// TwinCAT 3 PLC project MAS418
// ProgramVersion: 3.1.4023.0
// libraries:
//   Tc2_Standard, * (Beckhoff Automation GmbH)
//   Tc2_System, * (Beckhoff Automation GmbH)
//   Tc3_Module, * (Beckhoff Automation GmbH)
// project tree:
//   Actuators/FBs/ FB_AutoCyl.TcPOU, FB_autoWinch.TcPOU, FB_ClosedLoopControl.TcPOU, FB_Manual.TcPOU, FB_MotionReferenceGenerator.TcPOU, FB_OpenLoopControlCyl.TcPOU, FB_ResetIntegralController.TcPOU, FB_Timer.TcPOU, FB_OpenLoopWinchControl.TcPOU
//   Actuators/GVLs/ G_ControlParameters.TcGVL, G_Parameters.TcGVL
//   Actuators/Programs/ P_ControlSystem.TcPOU
//   Actuators/Structs/ ST_AutoControllerSelection.TcDUT, ST_ClosedLoopParams.TcDUT, ST_CylinderParameters.TcDUT, ST_MotionReferenceParams.TcDUT, ST_OpenLoopParams.TcDUT, ST_ScalingParameters.TcDUT, ST_SetControlParams.TcDUT, ST_ValveDeadband.TcDUT, ST_WinchParameters.TcDUT
//   / GlobalTextList.TcGTLO, PlcTask.TcTTO, Visualization Manager.TcVMO (not stored)
//   HMI/ CtrlBox.TcVIS, P_VHMI.TcPOU, VirtualBoxHMI.TcVIS
//   HMI/Enums/ E_Mode.TcDUT, E_Status.TcDUT, I_Mode.TcIO
//   HMI/FBs/ FB_Mode.TcPOU, FB_Status.TcPOU
//   HMI/GVLs/ G_Modes.TcGVL
//   HMI/Structs/ ST_VisuParam.TcDUT
//   Inputs/FBs/ FB_Encoder.TcPOU, FB_FlowScaling.TcPOU, FB_JoystickScale.TcPOU, FB_Scaling.TcPOU
//   Inputs/GVLs/ G_InputsRaw.TcGVL, G_InputsScaled.TcGVL, G_StructData.TcGVL
//   Inputs/Programs/ P_ScaleSensors.TcPOU
//   Inputs/Structs/ ST_FlowScale.TcDUT, ST_InputScaling.TcDUT, ST_JoystickScale.TcDUT
//   Outputs/FBs/ FB_ValveOutput.TcPOU
//   Outputs/GVLs/ G_Outputs.TcGVL
//   Outputs/Programs/ P_out.TcPOU
//   Outputs/Structs/ ST_ValveOutput.TcDUT
//   POUs/ MAIN.TcPOU
// real-time tasks:
//   TASK PlcTask: cycle T#10ms, priority 20, ADS port 350
// I/O:
//   DEVICE Device 1 (EtherCAT) (disabled), AmsNetId 169.254.36.244.2.1
//     Term 1 (EK1100) [EK1100 EtherCAT Coupler (2A E-Bus)]
//       Term 2 (EL1008)
//       Term 3 (EL2008)
//       Term 4 (EL3068)
//       Term 5 (EL3068) [EL3068 8Ch. Ana. Input 0-10V]
//       Term 6 (EL3174) [EL3174 4Ch. Ana. Input +/-10V Diff., +/-20mA SingleEnded, 16 Bit]
//       Term 7 (EL3255)
//       Term 8 (EL4104)
//       Term 9 (EL9011)
//     Box 10 (Fraba EtherCAT) [Absolute Rotary Encoder IXARC V01.05]
// variable links:
//   MAS418 Instance <-> Device 1 (EtherCAT)/Box 10 (Fraba EtherCAT)
//     PlcTask Inputs/G_InputsRaw.nEncoderValue <-> Encoder/Position Value
//   MAS418 Instance <-> Device 1 (EtherCAT)/Term 1 (EK1100)/Term 2 (EL1008)
//     PlcTask Inputs/G_InputsRaw.bJoyTopSwitch <-> Channel 5/Input
//     PlcTask Inputs/G_InputsRaw.bSelectAuto <-> Channel 2/Input
//     PlcTask Inputs/G_InputsRaw.bSelectManual <-> Channel 1/Input
//     PlcTask Inputs/G_InputsRaw.bStartButton <-> Channel 3/Input
//     PlcTask Inputs/G_InputsRaw.bStopButton <-> Channel 4/Input
//   MAS418 Instance <-> Device 1 (EtherCAT)/Term 1 (EK1100)/Term 3 (EL2008)
//     PlcTask Outputs/G_Outputs.bGreenLight <-> Channel 1/Output
//     PlcTask Outputs/G_Outputs.bRedLight <-> Channel 2/Output
//     PlcTask Outputs/G_Outputs.stCylinderOutputs.bEnable <-> Channel 4/Output
//     PlcTask Outputs/G_Outputs.stWinchOutputs.bEnable <-> Channel 3/Output
//   MAS418 Instance <-> Device 1 (EtherCAT)/Term 1 (EK1100)/Term 4 (EL3068)
//     PlcTask Inputs/G_InputsRaw.nPistonPressure <-> AI Standard Channel 4/Value
//     PlcTask Inputs/G_InputsRaw.nReturnPressure <-> AI Standard Channel 2/Value
//     PlcTask Inputs/G_InputsRaw.nRodPressure <-> AI Standard Channel 3/Value
//     PlcTask Inputs/G_InputsRaw.nSupplyPressure <-> AI Standard Channel 1/Value
//     PlcTask Inputs/G_InputsRaw.nWinch_A1_Pressure <-> AI Standard Channel 5/Value
//     PlcTask Inputs/G_InputsRaw.nWinch_A_Pressure <-> AI Standard Channel 7/Value
//     PlcTask Inputs/G_InputsRaw.nWinch_B1_Pressure <-> AI Standard Channel 6/Value
//     PlcTask Inputs/G_InputsRaw.nWinch_B_Pressure <-> AI Standard Channel 8/Value
//   MAS418 Instance <-> Device 1 (EtherCAT)/Term 1 (EK1100)/Term 5 (EL3068)
//     PlcTask Inputs/G_InputsRaw.nWinchDrainPressure <-> AI Standard Channel 1/Value
//   MAS418 Instance <-> Device 1 (EtherCAT)/Term 1 (EK1100)/Term 6 (EL3174)
//     PlcTask Inputs/G_InputsRaw.nWinchFlow <-> AI Standard Channel 1/Value
//   MAS418 Instance <-> Device 1 (EtherCAT)/Term 1 (EK1100)/Term 7 (EL3255)
//     PlcTask Inputs/G_InputsRaw.nJoyCyl <-> AI Standard Channel 2/Value
//     PlcTask Inputs/G_InputsRaw.nJoyWinch <-> AI Standard Channel 3/Value
//     PlcTask Inputs/G_InputsRaw.nPositionCylPiston <-> AI Standard Channel 1/Value
//   MAS418 Instance <-> Device 1 (EtherCAT)/Term 1 (EK1100)/Term 8 (EL4104)
//     PlcTask Outputs/G_Outputs.stCylinderOutputs.nValveOutput <-> AO Output Channel 2/Analog output
//     PlcTask Outputs/G_Outputs.stWinchOutputs.nValveOutput <-> AO Output Channel 1/Analog output

CONFIGURATION MAS418
    RESOURCE PLC ON TwinCAT3
        TASK PlcTask(INTERVAL := T#10ms, PRIORITY := 20);
        PROGRAM MAIN WITH PlcTask : MAIN;
    END_RESOURCE
END_CONFIGURATION

// ---- Actuators/Structs/ST_AutoControllerSelection.TcDUT
TYPE ST_AutoControllerSelection :
STRUCT
	bStartFeedForward : BOOL;
	bStartClosedLoop : BOOL;
	bEnableIntegral : BOOL; 
	
END_STRUCT
END_TYPE

// ---- Actuators/Structs/ST_ClosedLoopParams.TcDUT
TYPE ST_ClosedLoopParams :
STRUCT
	fProportionalGain: LREAL;
	fIntegralGain: LREAL;
	fMaxAllowableError : LREAL; 
END_STRUCT
END_TYPE

// ---- Actuators/Structs/ST_CylinderParameters.TcDUT
TYPE ST_CylinderParameters :
STRUCT
	fCylMaxSpeed : LREAL := 0.05; // m/s
END_STRUCT
END_TYPE

// ---- Actuators/Structs/ST_MotionReferenceParams.TcDUT
TYPE ST_MotionReferenceParams :
STRUCT
	fStartPosition_m: LREAL := 0.0;
	fStartVelocity_m: LREAL := 0.0;
	fPositionSetpoint_m: LREAL := 0.2;
	fVelocitySetpoint_m: LREAL := 0.02;
	fTimeBeforeStarting_s: LREAL := 1.5;
	fRampTime_s: LREAL := 2.0;
	fHoldPositionTime_s: LREAL := 4.0;
	
	// Saturation
	fMaxPosition 			: LREAL := 0.6;
	fMinPosition 			: LREAL := 0.0;
	fMaxVelocity 			: LREAL := 0.04;
	
	// Cycle time
	fCycleTime : LREAL := 0.001; // Same as matlab/simulink
END_STRUCT
END_TYPE

// ---- Actuators/Structs/ST_OpenLoopParams.TcDUT
TYPE ST_OpenLoopParams :
STRUCT
	fBoresideArea : LREAL;
	fAnnulusArea : LREAL; 
	fMaxFlow : LREAL; 
END_STRUCT
END_TYPE

// ---- Actuators/Structs/ST_ScalingParameters.TcDUT
TYPE ST_ScalingParameters :
STRUCT
	stCylPos : ST_InputScaling := (fMaxInputValue := 32295.0, fMinInputValue := 229.0, fMaxOutputValue := 0.5, fMinOutputValue := 0.0);
	stPressure400bar 	: ST_InputScaling := (fMaxInputValue := 32767.0, fMinInputValue := 0.0, fMaxOutputValue := 400.0, fMinOutputValue := 0.0);
	stPressure40bar 	: ST_InputScaling := (fMaxInputValue := 32767.0, fMinInputValue := 0.0, fMaxOutputValue := 40.0, fMinOutputValue := 0.0);
	stFlow : ST_FlowScale := (fMaxFlowInput := 32295.0, fMinFlowInput := 0.0, fNeutralFlowInput := 15450, fNeutralDeadband := 50.0, fMaxFlowOutput := 150.0, fMinFlowOutput := -150.0, fNeutralFlowOutput := 0.0);
END_STRUCT
END_TYPE

// ---- Actuators/Structs/ST_SetControlParams.TcDUT
TYPE ST_SetControlParams :
STRUCT
	stWinchControlClosedSettings : ST_ClosedLoopParams :=(fProportionalGain:=10, fIntegralGain:=5, fMaxAllowableError := 0.01);
	stCylControlCloesSettings : ST_ClosedLoopParams :=(fProportionalGain:=10, fIntegralGain:=5, fMaxAllowableError := 0.01);
	stWinchControlOpenSettings : ST_OpenLoopParams :=(fBoresideArea:=0.0033183, fAnnulusArea:=0.0023562, fMaxFlow:=150*0.5);
	stCylControlOpenSettings : ST_OpenLoopParams :=(fBoresideArea:=0, fAnnulusArea:=0, fMaxFlow:=150*0.5); 
END_STRUCT
END_TYPE

// ---- Actuators/Structs/ST_ValveDeadband.TcDUT
TYPE ST_ValveDeadband :
STRUCT
	fPosMax	: LREAL := 29490.0; 
	fPosMin	: LREAL := 20950.0; 
	fNegMin : LREAL := 18250.0; 
	fNegMax	: LREAL := 9830.0; 
END_STRUCT
END_TYPE

// ---- Actuators/Structs/ST_WinchParameters.TcDUT
TYPE ST_WinchParameters :
STRUCT
	fEncoderOffset : LREAL := 17574.8;
	fWinchDrumScaling : LREAL := 0.000744309;
	fWinchMotorDisplacement : LREAL := 32.0; 
	fWinchMaxSpeed : LREAL := 0.05; // rad/s
	
END_STRUCT
END_TYPE

// ---- HMI/Enums/E_Mode.TcDUT
{attribute 'qualified_only'}
{attribute 'strict'}
TYPE E_Mode :
(
	OFF := 0,
	Auto := 1,
	Manual :=2
);
END_TYPE

// ---- HMI/Enums/E_Status.TcDUT
{attribute 'qualified_only'}
{attribute 'strict'}
TYPE E_Status :
(	NotReady := 0,
	Ready := 1,
	Starting := 2,
	Running := 3,
	Stopping := 4,
	Fault := 5,
	JoyStick := 6
);
END_TYPE

// ---- HMI/Structs/ST_VisuParam.TcDUT
TYPE ST_VisuParam :
STRUCT
bOn : BOOL;
bAuto : BOOL;
bStart : BOOL;
bStop : BOOL;
bRunning : BOOL;
bFault : BOOL;
fJoy_X : REAL;
fJoy_Y : REAL;
bTopSwitchJoy : BOOL;
END_STRUCT
END_TYPE

// ---- Inputs/Structs/ST_FlowScale.TcDUT
TYPE ST_FlowScale :
STRUCT
	fMaxFlowInput : LREAL; 
	fMinFlowInput : LREAL;
    fNeutralFlowInput : LREAL; 
	fNeutralDeadband : LREAL; 
	fMaxFlowOutput : LREAL; 
	fMinFlowOutput : LREAL; 
	fNeutralFlowOutput : LREAL; 
END_STRUCT
END_TYPE

// ---- Inputs/Structs/ST_InputScaling.TcDUT
TYPE ST_InputScaling :
STRUCT
	fMaxInputValue : LREAL;
	fMinInputValue : LREAL;
	fMaxOutputValue : LREAL;
	fMinOutputValue : LREAL; 
END_STRUCT
END_TYPE

// ---- Inputs/Structs/ST_JoystickScale.TcDUT
TYPE ST_JoystickScale :
STRUCT
	fMaxInputValue : LREAL := 20509.0;
	fMinInputValue : LREAL  := 11787.0; 
	fNeutralInputValue : LREAL  := 16175; 
	fNeutralDeadband : LREAL  := 50.0; 
	fMaxOutputValue : LREAL  := 1.0; 
	fMinOutputValue : LREAL  := -1.0;
	fNeutralOutputValue : LREAL  := 0.0; 
END_STRUCT
END_TYPE

// ---- Outputs/Structs/ST_ValveOutput.TcDUT
TYPE ST_ValveOutput :
STRUCT
	bEnable					AT %Q* : BOOL := 0;
	nValveOutput 			AT %Q* : INT := 19660; // Initial value at offset
END_STRUCT
END_TYPE

// ---- Actuators/GVLs/G_ControlParameters.TcGVL
{attribute 'qualified_only'}
VAR_GLOBAL
	bWinchEnable : BOOL;
	bCylEnable : BOOL;
	
	// Parameters for control circuit
	fWinch_ControlInput : LREAL;
	fWinchTimer	: LREAL;
	fCylinder_ControlInput : LREAL;
	fCylTimer : LREAL;
	fControlSignal_Winch : LREAL;
	fControlSignal_Cyl : LREAL; 
	
	// Reference signals / Setpoints
	fVelRefWinch : LREAL;
	fPosRefWinch : LREAL;
	fVelRefCyl : LREAL;
	fPosRefCyl : LREAL;
	fPosErrorWinch : LREAL;
	fPosErrorCyl : LREAL; 
	
	bDeadBandCompOn : BOOL := TRUE; 
END_VAR

// ---- Actuators/GVLs/G_Parameters.TcGVL
{attribute 'qualified_only'}
VAR_GLOBAL
	stCylParams : ST_CylinderParameters;
	stValve : ST_ValveDeadband;
	stWinchParams : ST_WinchParameters; 
	stCommonScaling : ST_ScalingParameters; 
	stControl : ST_SetControlParams;  
END_VAR

// ---- HMI/GVLs/G_Modes.TcGVL
{attribute 'qualified_only'}
VAR_GLOBAL
	bManualMode : BOOL;
	bAutoMode : BOOL; 
	bStart : BOOL;
	bStop : BOOL;
	bSwitch : BOOL; 
	bCylEnable : BOOL;
	bWinchEnable : BOOL; 
	bOn : BOOL; 
	stMotionRefWinch : ST_MotionReferenceParams;
	stMotionRefCyl : ST_MotionReferenceParams;
	stCylinderControl : ST_AutoControllerSelection;
	stWinchControl : ST_AutoControllerSelection; 
	eStatus : E_Status;
	eMode : E_Mode; 
	stVisualParams : ST_VisuParam; 
END_VAR

// ---- Inputs/GVLs/G_InputsRaw.TcGVL
{attribute 'qualified_only'}
VAR_GLOBAL
	bSelectOff AT %I* : BOOL; 
	bSelectManual	AT %I* : BOOL;
	bSelectAuto AT %I* : BOOL;
	bStartButton AT %I* : BOOL;
	bStopButton	AT %I* : BOOL;
	bJoyTopSwitch	AT %I* : BOOL;
	
	// Joystick
	nJoyCyl AT %I* : INT; 					
	nJoyWinch AT %I* : INT; 	

	// Encoder					
	nPositionCylPiston AT %I* : INT; 		
	nEncoderValue AT %I* : UDINT;
		
	
	// Pressures Valve x Cyl
	nSupplyPressure AT %I* : INT;
	nReturnPressure AT %I* : INT;
	nPistonPressure AT %I* : INT;
	nRodPressure AT %I* : INT; 
	
	// Pressures Winch
	nWinch_A_Pressure AT %I* : INT;
	nWinch_A1_Pressure AT %I* : INT;
	nWinch_B_Pressure AT %I* : INT;
	nWinch_B1_Pressure AT %I* : INT;
	nWinchDrainPressure AT %I* : INT; 

	// Winch flow
	nWinchFlow AT %I* : INT; 		
END_VAR

// ---- Inputs/GVLs/G_InputsScaled.TcGVL
{attribute 'qualified_only'}
VAR_GLOBAL
	
	// Joystick
	fJoystickScaledX 		: LREAL;
	fJoystickScaledY 		: LREAL;
	
	// Cylinder and winch position
	fCylPosition : LREAL;	
	fEncoderPosition : LREAL;
	fWirePosition : LREAL;
	
	// Pressures Valve
	fSupplyPressure			: LREAL;
	fReturnPressure 			: LREAL;
	
	// Pressures Cylinder
	fPistonPressure 	: LREAL;
	fRodPressure		: LREAL;
	
	// Pressures Winch
	fWinch_A_Pressure 		: LREAL;
	fWinch_A1_Pressure 		: LREAL;
	fWinch_B_Pressure	: LREAL;
	fWinch_B1_Pressure	: LREAL;
	fWinchDrainPressure			: LREAL;
	
	// Winch Flow
	fWinchFlow 					: LREAL;
END_VAR

// ---- Inputs/GVLs/G_StructData.TcGVL
{attribute 'qualified_only'}
VAR_GLOBAL
	stJoystickX : ST_JoystickScale;
	stJoystickY : ST_JoystickScale; 
	stInputs : ST_InputScaling;
	stFlows : ST_FlowScale;
END_VAR

// ---- Outputs/GVLs/G_Outputs.TcGVL
{attribute 'qualified_only'}
VAR_GLOBAL
	bGreenLight AT %Q* : BOOL;
	bRedLight AT %Q* : BOOL;
	
	stWinchOutputs : ST_ValveOutput;
	stCylinderOutputs : ST_ValveOutput; 
END_VAR

// ---- HMI/Enums/I_Mode.TcIO

INTERFACE I_Mode

METHOD Auto
VAR_INPUT
	bEnable : BOOL;
END_VAR
END_METHOD

METHOD Manual
VAR_INPUT
	bEnable : BOOL;
END_VAR
END_METHOD

METHOD OFF 
VAR_INPUT
	bEnable : BOOL;
END_VAR
END_METHOD

END_INTERFACE

// ---- POUs/MAIN.TcPOU
PROGRAM MAIN
VAR
END_VAR

P_ScaleSensors();
P_out();
P_VHMI();
P_ControlSystem();

END_PROGRAM

// ---- Inputs/Programs/P_ScaleSensors.TcPOU
PROGRAM P_ScaleSensors
VAR
	// Joystick
	fbJoystickX : FB_JoystickScale;
	fbJoystickY : FB_JoystickScale;
	
	// Positions
	fbWinchPosition : FB_Encoder;
	fbCylPosition : FB_Scaling;
	
	// Pressures
	fbSupplyPressure : FB_Scaling;
	fbReturnPressure : FB_Scaling;
	fbPistonPressure : FB_Scaling;
	fbRodPressure	: FB_Scaling;
	fbWinch_A_Pressure : FB_Scaling;
	fbWinch_A1_Pressure : FB_Scaling;
	fbWinch_B_Pressure : FB_Scaling;
	fbWinch_B1_Pressure : FB_Scaling;
	fbWinchDrainPressure : FB_Scaling;
	
	// Flows
	fbWinchFlow	: FB_FlowScaling;
END_VAR

// Scaling Joystick
fbJoystickX(bEnable := G_Modes.bManualMode, nRawInput := G_InputsRaw.nJoyCyl,
	fNormalizedOutput => G_InputsScaled.fJoystickScaledX);

fbJoystickY(bEnable := G_Modes.bManualMode, 
	nRawInput := G_InputsRaw.nJoyWinch, 
	fNormalizedOutput => G_InputsScaled.fJoystickScaledY);
 
// Winch position & Cylinder position
fbWinchPosition (
	nRawInput := G_InputsRaw.nEncoderValue, 
	fPosition => G_InputsScaled.fEncoderPosition,
	fWirePosition => G_InputsScaled.fWirePosition);

fbCylPosition(
	nRawInput := G_InputsRaw.nPositionCylPiston,
	stInputScaling := G_Parameters.stCommonScaling.stCylPos,
	fScaledOutput => G_InputsScaled.fCylPosition);


// Pressures

fbSupplyPressure(
	nRawInput := G_InputsRaw.nSupplyPressure,
	stInputScaling := G_Parameters.stCommonScaling.stPressure400bar,
	fScaledOutput => G_InputsScaled.fSupplyPressure);

fbReturnPressure(
	nRawInput := G_InputsRaw.nReturnPressure,
	stInputScaling := G_Parameters.stCommonScaling.stPressure40bar,
	fScaledOutput => G_InputsScaled.fReturnPressure);

fbPistonPressure(
	nRawInput := G_InputsRaw.nPistonPressure,
	stInputScaling := G_Parameters.stCommonScaling.stPressure400bar,
	fScaledOutput => G_InputsScaled.fPistonPressure);
	
fbRodPressure(
	nRawInput := G_InputsRaw.nRodPressure,
	stInputScaling := G_Parameters.stCommonScaling.stPressure400bar,
	fScaledOutput => G_InputsScaled.fRodPressure);
	
fbWinch_A_Pressure(
	nRawInput := G_InputsRaw.nWinch_A_Pressure,
	stInputScaling := G_Parameters.stCommonScaling.stPressure400bar,
	fScaledOutput => G_InputsScaled.fWinch_A_Pressure); 
	
fbWinch_A1_Pressure(
	nRawInput := G_InputsRaw.nWinch_A1_Pressure,
	stInputScaling := G_Parameters.stCommonScaling.stPressure400bar,
	fScaledOutput => G_InputsScaled.fWinch_A1_Pressure);

fbWinch_B_Pressure(
	nRawInput := G_InputsRaw.nWinch_B_Pressure,
	stInputScaling := G_Parameters.stCommonScaling.stPressure400bar,
	fScaledOutput => G_InputsScaled.fWinch_B_Pressure);

fbWinch_B1_Pressure(
	nRawInput := G_InputsRaw.nWinch_B1_Pressure,
	stInputScaling := G_Parameters.stCommonScaling.stPressure400bar,
	fScaledOutput => G_InputsScaled.fWinch_B1_Pressure);
	
fbWinchDrainPressure(
	nRawInput := G_InputsRaw.nWinchDrainPressure,
	stInputScaling := G_Parameters.stCommonScaling.stPressure40bar,
	fScaledOutput => G_InputsScaled.fWinchDrainPressure);

fbWinchFlow(
	nRawInput := G_InputsRaw.nWinchFlow,
	stFlowParams := G_Parameters.stCommonScaling.stFlow,
	fScaledFlow => G_InputsScaled.fWinchFlow);

END_PROGRAM

// ---- Inputs/FBs/FB_JoystickScale.TcPOU
FUNCTION_BLOCK FB_JoystickScale
VAR_INPUT
	bEnable 				: BOOL;
	nRawInput 				: INT;
END_VAR
VAR_OUTPUT
	fNormalizedOutput 		: LREAL;
END_VAR
VAR
	stJoystickScale  : ST_JoystickScale;
	fRawInput 				: LREAL;
	fTempInput 				: LREAL;
	fTempOutput 			: LREAL;
END_VAR

fRawInput := INT_TO_LREAL(nRawInput);

fTempInput := fRawInput - stJoystickScale.fNeutralInputValue;

IF fTempInput > stJoystickScale.fNeutralDeadband THEN
	fTempOutput := fTempInput/(stJoystickScale.fMaxInputValue - stJoystickScale.fNeutralInputValue);
ELSIF fTempInput < -stJoystickScale.fNeutralDeadband THEN	
	fTempOutput := fTempInput/(stJoystickScale.fNeutralInputValue - stJoystickScale.fMinInputValue);
ELSE
	fTempOutput := 0.0;
END_IF

IF NOT(bEnable) THEN
	fNormalizedOutput := 0.0;
ELSE
	fNormalizedOutput := LIMIT(stJoystickScale.fMinOutputValue, fTempOutput, stJoystickScale.fMaxOutputValue);
END_IF

END_FUNCTION_BLOCK

// ---- Inputs/FBs/FB_Encoder.TcPOU
FUNCTION_BLOCK FB_Encoder
VAR_INPUT
	nRawInput : UDINT;
	stParam 		: ST_WinchParameters; 
END_VAR
VAR_OUTPUT
	fPosition 		: LREAL;
	fWirePosition : LREAL; 
END_VAR
VAR PERSISTENT
	nRounds			: DINT;
	nRawLast 		: DINT;
END_VAR	
VAR
	nInput 		: DINT;
	nTempInputDiff	: DINT;
	nCount 			: DINT;
	nMaxValue30bit 	: DINT :=  1073741823; // 2^30 - 1	
	nThreshold30bit	: DINT := nMaxValue30bit/2;
	fScale16bit		: LREAL := 360.0/65535.0; // 360deg/(2^16 - 1)
	fTempPosition   : LREAL;
END_VAR

// Convert to DINT (same as const values)
nInput := UDINT_TO_DINT(nRawInput);

// Define Encoder Rounds
nTempInputDiff := nInput - nRawLast;
IF (nTempInputDiff > nThreshold30bit) THEN
	nRounds := nRounds - 1;
END_IF

IF (nTempInputDiff < -nThreshold30bit) THEN
	nRounds := nRounds + 1;
END_IF

// Count Encoder Rounds
nCount := nInput + nRounds*nMaxValue30bit;

//Position Output
fPosition := DINT_TO_LREAL(nCount)*fScale16bit - stParam.fEncoderOffset; // Encoder position
fWirePosition := fPosition * G_Parameters.stWinchParams.fWinchDrumScaling; // WIre position

END_FUNCTION_BLOCK

// ---- Inputs/FBs/FB_Scaling.TcPOU
FUNCTION_BLOCK FB_Scaling
VAR_INPUT
	nRawInput : INT; 
	stInputScaling : ST_InputScaling; 
END_VAR
VAR_OUTPUT
	fScaledOutput : LREAL;

END_VAR
VAR
	fRawInput : LREAL;
	fNormInput : LREAL;
	
END_VAR

fRawInput := INT_TO_LREAL(nRawInput);

fNormInput := (fRawInput - stInputScaling.fMinInputValue) / (stInputScaling.fMaxInputValue - stInputScaling.fMinInputValue);

fScaledOutput := LIMIT(stInputScaling.fMinOutputValue, stInputScaling.fMinOutputValue + fNormInput*(stInputScaling.fMaxOutputValue - stInputScaling.fMinOutputValue), stInputScaling.fMaxOutputValue);

END_FUNCTION_BLOCK

// ---- Inputs/FBs/FB_FlowScaling.TcPOU
FUNCTION_BLOCK FB_FlowScaling
VAR_INPUT
	nRawInput : INT;
	stFlowParams : ST_FlowScale; 
END_VAR
VAR_OUTPUT
	fScaledFlow : LREAL; 
END_VAR
VAR
	fRawInput 				: LREAL;
	fTempInput 				: LREAL;
	fTempOutput 			: LREAL;
END_VAR

fRawInput := INT_TO_LREAL(nRawInput);

fTempInput := fRawInput - stFlowParams.fNeutralFlowInput;

IF fTempInput > stFlowParams.fNeutralDeadband THEN
	fTempOutput := fTempInput/(stFlowParams.fMaxFlowInput - stFlowParams.fNeutralFlowInput);
ELSIF fTempInput < -stFlowParams.fNeutralDeadband THEN	
	fTempOutput := fTempInput/(stFlowParams.fNeutralFlowInput - stFlowParams.fMinFlowInput);
ELSE
	fTempOutput := 0.0;
END_IF

fScaledFlow := LIMIT(stFlowParams.fMinFlowOutput, fTempOutput*150.0, stFlowParams.fMaxFlowOutput);

END_FUNCTION_BLOCK

// ---- Outputs/Programs/P_out.TcPOU
PROGRAM P_out
VAR
	fbWinchOutput 		: FB_ValveOutput;
	fbCylOutput 		: FB_ValveOutput;
END_VAR

// Settings to ensure output if either auto or manual is selected:
G_Outputs.stWinchOutputs.bEnable := G_Modes.bAutoMode OR G_Modes.bManualMode; 
G_Outputs.stCylinderOutputs.bEnable := G_Modes.bAutoMode OR G_Modes.bManualMode; 


fbWinchOutput(bEnable := G_ControlParameters.bWinchEnable OR G_ControlParameters.fWinchTimer > 0.0,
	bDeadBandCompOn := G_ControlParameters.bDeadBandCompOn,
	stValveDeadBand := G_Parameters.stValve,
	fNormalizedInput := G_ControlParameters.fWinch_ControlInput,
	nOutput => G_Outputs.stWinchOutputs.nValveOutput); 
	
	
fbCylOutput(bEnable := G_ControlParameters.bWinchEnable OR G_ControlParameters.fCylTimer > 0.0,
	bDeadBandCompOn := G_ControlParameters.bDeadBandCompOn,
	stValveDeadBand := G_Parameters.stValve,
	fNormalizedInput := G_ControlParameters.fCylinder_ControlInput,
	nOutput => G_Outputs.stCylinderOutputs.nValveOutput);

END_PROGRAM

// ---- Outputs/FBs/FB_ValveOutput.TcPOU
FUNCTION_BLOCK FB_ValveOutput
VAR_INPUT
	bEnable 			: BOOL;
	bDeadBandCompOn 	: BOOL;
	stValveDeadBand 	: ST_ValveDeadBand;
	fNormalizedInput 	: LREAL;
END_VAR
VAR_OUTPUT
	bEnableValveOutput : BOOL;
	nOutput : INT; 
END_VAR
VAR
	nOffset 	: INT := 19660;
	nMaxValue	: INT := 29490;
	nMinValue 	: INT :=  9830;
	nTempOutput : INT;
END_VAR

IF	bDeadBandCompOn THEN
	IF fNormalizedInput > 0.0 THEN
		nTempOutput := LREAL_TO_INT(ABS(fNormalizedInput*(stValveDeadBand.fPosMax - stValveDeadBand.fPosMin) + stValveDeadBand.fPosMin));
	ELSIF fNormalizedInput < 0.0 THEN
		nTempOutput := LREAL_TO_INT(ABS(fNormalizedInput*(stValveDeadBand.fNegMax - stValveDeadBand.fNegMin) - stValveDeadBand.fNegMin));
	ELSE
		nTempOutput := nOffset;
	END_IF
ELSE
	IF fNormalizedInput > 0.0 THEN
		nTempOutput := LREAL_TO_INT(ABS(fNormalizedInput*(32767.0 - 19660.0) + 19660.0));
	ELSIF fNormalizedInput < 0.0 THEN
		nTempOutput := LREAL_TO_INT(ABS(fNormalizedInput*(0 - 19660.0) - 19660.0));
	ELSE
		nTempOutput := nOffset;
	END_IF	
END_IF	

IF bEnable THEN
	nOutput := LIMIT(nMinValue, nTempOutput, nMaxValue);
	bEnableValveOutput := TRUE; 
ELSE 	
	nOutput := nOffset;
	bEnableValveOutput := FALSE;	
END_IF

END_FUNCTION_BLOCK

// ---- HMI/P_VHMI.TcPOU
PROGRAM P_VHMI
VAR
	fbModeSelect : FB_Mode;
END_VAR

fbModeSelect(
	bMode := G_Modes.bAutoMode);

END_PROGRAM

// ---- HMI/FBs/FB_Mode.TcPOU
FUNCTION_BLOCK FB_Mode
VAR_INPUT
	bMode : BOOL; 
END_VAR
VAR_OUTPUT
	
END_VAR
VAR
END_VAR

IF bMode THEN
	G_Modes.eMode := E_Mode.Auto;
ELSIF NOT bMode AND NOT G_Modes.bOn THEN
	G_Modes.eMode := E_Mode.OFF;
ELSE
	G_Modes.eMode := E_Mode.Manual;
END_IF

END_FUNCTION_BLOCK

// ---- Actuators/Programs/P_ControlSystem.TcPOU
PROGRAM P_ControlSystem
VAR
	fbManualWinchControl : FB_Manual;
	fbManualCylinderControl : FB_Manual; 
	fbAutoWinchControl : FB_autoWinch;
	fbAutoCylinderControl : FB_AutoCyl; 
	
	fWinchManualSignal : LREAL;
	fCylManualSignal : LREAL; 
	
END_VAR

G_Modes.bAutoMode := G_InputsRaw.bSelectAuto;
G_Modes.bManualMode := G_InputsRaw.bSelectManual; 
G_Modes.bSwitch := G_InputsRaw.bJoyTopSwitch; 
G_ControlParameters.bCylEnable := G_Modes.bCylEnable;
G_ControlParameters.bWinchEnable := G_Modes.bWinchEnable; 

fbManualCylinderControl(
	bEnable := G_Modes.bManualMode AND G_InputsRaw.bStartButton AND NOT G_Modes.bSwitch,
	fInput := G_InputsScaled.fJoystickScaledX,
	fControlRefSignal => fCylManualSignal
); 

fbManualWinchControl(
	bEnable := G_Modes.bManualMode AND G_Modes.bSwitch AND G_InputsRaw.bStartButton,
	fInput := G_InputsScaled.fJoystickScaledY,
	fControlRefSignal => fWinchManualSignal
); 

fbAutoWinchControl(
	bEnable := G_Modes.bAutoMode AND G_ControlParameters.bWinchEnable,
	bStartMotion := G_InputsRaw.bStartButton,
	bStopMotion := G_InputsRaw.bStopButton,
	stMotionRefGenerator := G_Modes.stMotionRefWinch,
	stClosedLoopControl := G_Parameters.stControl.stWinchControlClosedSettings,
	stOpenLoopControl := G_Parameters.stControl.stWinchControlOpenSettings,
	stControlSelect := G_Modes.stWinchControl,
	stScaledValues := G_Parameters.stCommonScaling,
	//stScaledWinch := G_Parameters.stCommonScaling,
	fPositionFeedback := G_InputsScaled.fWirePosition,
	fTime => G_ControlParameters.fWinchTimer,
	fVelocityReference_ms => G_ControlParameters.fVelRefWinch,
	fPositionReference_m => G_ControlParameters.fPosRefWinch,
	fControlOutputNormalized => G_ControlParameters.fControlSignal_Winch,
	fPositionError_mm => G_ControlParameters.fPosErrorWinch); 
	
fbAutoCylinderControl(
	bEnable := G_Modes.bAutoMode AND G_ControlParameters.bCylEnable,
	bStartMotion := G_InputsRaw.bStartButton,
	bStopMotion := G_InputsRaw.bStopButton,
	stMotionRefGenerator := G_Modes.stMotionRefCyl,
	stClosedLoopControl := G_Parameters.stControl.stCylControlCloesSettings,
	stOpenLoopControl := G_Parameters.stControl.stCylControlOpenSettings,
	stControlSelect := G_Modes.stCylinderControl,
	stScaledValues := G_Parameters.stCommonScaling,
	//stScaledWinch := G_Parameters.stCommonScaling,
	fPositionFeedback := G_InputsScaled.fCylPosition,
	fTime => G_ControlParameters.fCylTimer,
	fVelocityReference_ms => G_ControlParameters.fVelRefCyl,
	fPositionReference_m => G_ControlParameters.fPosRefCyl,
	fControlOutputNormalized => G_ControlParameters.fControlSignal_Cyl,
	fPositionError_mm => G_ControlParameters.fPosErrorCyl); 

IF G_Modes.bManualMode THEN
	G_ControlParameters.fCylinder_ControlInput := fCylManualSignal;
	G_ControlParameters.fWinch_ControlInput := fWinchManualSignal;
ELSIF G_Modes.bAutoMode THEN
	G_ControlParameters.fCylinder_ControlInput := G_ControlParameters.fControlSignal_Cyl;
	G_ControlParameters.fWinch_ControlInput := G_ControlParameters.fControlSignal_Winch;
	
ELSE
	G_ControlParameters.fCylinder_ControlInput := 0.0;
	G_ControlParameters.fWinch_ControlInput := 0.0; 
END_IF

END_PROGRAM

// ---- Actuators/FBs/FB_Manual.TcPOU
FUNCTION_BLOCK FB_Manual
VAR_INPUT
	bEnable : BOOL;
	fInput : LREAL;

END_VAR
VAR_OUTPUT
	fControlRefSignal	: LREAL;
END_VAR
VAR
END_VAR

IF NOT(bEnable) THEN
	fControlRefSignal := 0.0; 
ELSE
	fControlRefSignal := fInput;
END_IF

END_FUNCTION_BLOCK

// ---- Actuators/FBs/FB_autoWinch.TcPOU
FUNCTION_BLOCK FB_autoWinch
VAR_INPUT
	bEnable 							: BOOL;
	bStartMotion 						: BOOL;
	bStopMotion 						: BOOL;
	stMotionRefGenerator : ST_MotionReferenceParams;
	stClosedLoopControl : ST_ClosedLoopParams;
	stOpenLoopControl : ST_OpenLoopParams;
	stControlSelect			: ST_AutoControllerSelection;
	stScaledValues : ST_ScalingParameters;
	stScaledWinch : ST_WinchParameters;  
	fPositionFeedback					: LREAL;
END_VAR
VAR_OUTPUT
	fTime : LREAL;
	fVelocityReference_ms : LREAL;
	fPositionReference_m : LREAL;
	fControlOutputNormalized : LREAL;
	fPositionError_mm : LREAL;
END_VAR
VAR
	fbClock : FB_Timer;	
	fbMotionReferenceGenerator 		: FB_MotionReferenceGenerator;	
	fbFeedForwardControl 	: FB_OpenLoopWinchControl;
	fbResetIntegralController 		: FB_ResetIntegralController; 
	fbClosedLoopControl 	: FB_ClosedLoopControl;
END_VAR

fbClock(
	bEnable := bEnable,
	bStart := bStartMotion,
	bStop := bStopMotion,
	fCycleTime := stMotionRefGenerator.fCycleTime);

fbMotionReferenceGenerator(
	bEnable := bEnable,
	stMotionParameters := stMotionRefGenerator,
	fClock_s := fbClock.fTime);

fbFeedForwardControl(
	bEnable := stControlSelect.bStartFeedForward,
	fVelocityReference_ms := fbMotionReferenceGenerator.fVelocityReference_m,
	stOpenLoopSettings := stOpenLoopControl); 
	
fbResetIntegralController(
	fMaxPositionError_m := stClosedLoopControl.fMaxAllowableError,
	fPositionError_m := fbClosedLoopControl.fPositionError,
	fVelocityReference_ms := fbMotionReferenceGenerator.fVelocityReference_m
	
); 

fbClosedLoopControl(
	bEnable := stControlSelect.bStartClosedLoop,
	bActivateIntegralController := stControlSelect.bEnableIntegral,
	fPositionReference := fbMotionReferenceGenerator.fPositionReference_m,
	fPositionFeedback := fPositionFeedback,
	bIntegralControllReset := fbResetIntegralController.bReset,
	stClosedLoopParams := stClosedLoopControl,
	stMotionParams := stMotionRefGenerator
	
);

fVelocityReference_ms := fbMotionReferenceGenerator.fVelocityReference_m;
fPositionReference_m := fbMotionReferenceGenerator.fPositionReference_m;
fTime := fbClock.fTime;
fPositionError_mm := fbClosedLoopControl.fPositionError*1E3; 

IF bEnable THEN
	fControlOutputNormalized := LIMIT(-1.0, (fbFeedForwardControl.fOutput + fbClosedLoopControl.fClosedLoopPosition), 1.0); 
ELSE
	fControlOutputNormalized := 0.0; 
END_IF

END_FUNCTION_BLOCK

// ---- Actuators/FBs/FB_Timer.TcPOU
FUNCTION_BLOCK FB_Timer
VAR_INPUT
	bEnable 	: BOOL;
	bStart 		: BOOL;
	bStop 		: BOOL;
	fCycleTime  : LREAL;
END_VAR
VAR_OUTPUT
	fTime : LREAL;
END_VAR
VAR
END_VAR

IF bStart AND NOT(bStop) AND bEnable THEN
	fTime := fTime + fCycleTime;
ELSE
	fTime := 0.0;
END_IF

END_FUNCTION_BLOCK

// ---- Actuators/FBs/FB_MotionReferenceGenerator.TcPOU
FUNCTION_BLOCK FB_MotionReferenceGenerator
VAR_INPUT
	bEnable: BOOL;
	stMotionParameters : ST_MotionReferenceParams;
	fClock_s: LREAL;
END_VAR
VAR_OUTPUT
	fPositionReference_m: LREAL;
	fVelocityReference_m: LREAL;
	fTotalMotionTime_s: LREAL;
	bErrorSignal: BOOL;
END_VAR
VAR
	fStartPosition_m		: LREAL;
	fStartVelocity_m		: LREAL;
	fPositionSetpoint_ms	: LREAL;
	fVelocitySetpoint_m		: LREAL;
	fTimeBeforeStarting_s	: LREAL;
	fRampTime_s				: LREAL;
	fHoldPositionTime_s		: LREAL;
	Error: DINT;
	slopeExt: LREAL;
	slopeRetr : LREAL;
	tHold: LREAL;
	x1: LREAL;
	x4: LREAL;
	x1_tmp: LREAL;
	x1_tmp_tmp: LREAL;
	x4_tmp: LREAL;
	x4_tmp_tmp: LREAL;
	x4_tmp_tmp_0: LREAL;
	x4_tmp_tmp_1: LREAL;
	x1_tmp_0: LREAL;
END_VAR


// Saturating
fStartPosition_m := LIMIT(stMotionParameters.fMinPosition, stMotionParameters.fStartPosition_m, stMotionParameters.fMaxPosition);
fStartVelocity_m := LIMIT(0.0, stMotionParameters.fStartVelocity_m, stMotionParameters.fMaxVelocity);
fPositionSetpoint_ms := LIMIT(stMotionParameters.fMinPosition, stMotionParameters.fPositionSetpoint_m, stMotionParameters.fMaxPosition);
fVelocitySetpoint_m := LIMIT(0.0, stMotionParameters.fVelocitySetpoint_m, stMotionParameters.fMaxVelocity);
fTimeBeforeStarting_s := LIMIT(0.0, stMotionParameters.fTimeBeforeStarting_s, 10.0);
fRampTime_s := LIMIT(0.0, stMotionParameters.fRampTime_s, 10.0);
fHoldPositionTime_s := LIMIT(0.0, stMotionParameters.fHoldPositionTime_s, 60.0);

// Start of path
slopeExt := fStartVelocity_m - fVelocitySetpoint_m;
slopeRetr := ( -fVelocitySetpoint_m) - fStartVelocity_m;
tHold := ((fPositionSetpoint_ms - fStartPosition_m) - (((fVelocitySetpoint_m * fVelocitySetpoint_m) - (fStartVelocity_m * fStartVelocity_m)) / (fVelocitySetpoint_m / fRampTime_s))) / fVelocitySetpoint_m;


IF tHold < 0.0  THEN 
    bErrorSignal := TRUE;
ELSE 
    bErrorSignal := FALSE;
END_IF;
x1_tmp_tmp := fTimeBeforeStarting_s + fRampTime_s;
x1_tmp := x1_tmp_tmp - fTimeBeforeStarting_s;
x1_tmp_0 := slopeExt / fRampTime_s;
x1 := ((x1_tmp * fStartVelocity_m) + fStartPosition_m) - ((x1_tmp_0 * (x1_tmp * x1_tmp)) / 2.0);
x4_tmp_tmp := x1_tmp_tmp + tHold;
x4_tmp_tmp_0 := x4_tmp_tmp + fRampTime_s;
x4_tmp := x4_tmp_tmp_0 + fHoldPositionTime_s;
x1_tmp := x4_tmp + fRampTime_s;
x4 := x1_tmp - x4_tmp;
x4 := (fPositionSetpoint_ms - (x4 * fStartVelocity_m)) + (((slopeRetr / fRampTime_s) * (x4 * x4)) / 2.0);
IF Error = 1 THEN 
    fPositionReference_m := fStartPosition_m;
    fVelocityReference_m := fStartVelocity_m;
ELSIF (fClock_s >= 0.0) AND (fClock_s < fTimeBeforeStarting_s) THEN 
    fPositionReference_m := fStartPosition_m;
    fVelocityReference_m := fStartVelocity_m;
ELSIF (fClock_s >= fTimeBeforeStarting_s) AND (fClock_s < x1_tmp_tmp) THEN 
    slopeRetr := fClock_s - fTimeBeforeStarting_s;
    fPositionReference_m := ((slopeRetr * fStartVelocity_m) + fStartPosition_m) - ((x1_tmp_0 * (slopeRetr * slopeRetr)) / 2.0);
    fVelocityReference_m := fStartVelocity_m - (x1_tmp_0 * slopeRetr);
ELSIF (fClock_s >= x1_tmp_tmp) AND (fClock_s < x4_tmp_tmp) THEN 
    fPositionReference_m := ((fClock_s - x1_tmp_tmp) * fVelocitySetpoint_m) + x1;
    fVelocityReference_m := fVelocitySetpoint_m;
ELSIF (fClock_s >= x4_tmp_tmp) AND (fClock_s < x4_tmp_tmp_0) THEN 
    slopeRetr := fClock_s - x4_tmp_tmp;
    fPositionReference_m := ((((x4_tmp_tmp - x1_tmp_tmp) * fVelocitySetpoint_m) + x1) + (slopeRetr * fVelocitySetpoint_m)) + ((x1_tmp_0 * (slopeRetr * slopeRetr)) / 2.0);
    fVelocityReference_m := (slopeRetr * (slopeExt / fRampTime_s)) + fVelocitySetpoint_m;
ELSIF (fClock_s >= x4_tmp_tmp_0) AND (fClock_s < x4_tmp) THEN 
    fPositionReference_m := fPositionSetpoint_ms;
    fVelocityReference_m := fStartVelocity_m;
ELSIF (fClock_s >= x4_tmp) AND (fClock_s < x1_tmp) THEN 
    slopeExt := fClock_s - x4_tmp;
    slopeRetr := slopeRetr / fRampTime_s;
    fPositionReference_m := (fPositionSetpoint_ms - (slopeExt * fStartVelocity_m)) + ((slopeRetr * (slopeExt * slopeExt)) / 2.0);
    fVelocityReference_m := (slopeExt * slopeRetr) + fStartVelocity_m;
ELSE 
    x1_tmp_0 := x1_tmp + tHold;
    IF (fClock_s >= x1_tmp) AND (fClock_s < x1_tmp_0) THEN 
        fPositionReference_m := x4 - ((fClock_s - x1_tmp) * fVelocitySetpoint_m);
        fVelocityReference_m :=  -fVelocitySetpoint_m;
    ELSIF (fClock_s >= x1_tmp_0) AND (fClock_s < (((((((fTimeBeforeStarting_s + fRampTime_s) + tHold) + fRampTime_s) + fHoldPositionTime_s) + fRampTime_s) + tHold) + fRampTime_s)) THEN 
        slopeExt := fClock_s - x1_tmp_0;
        slopeRetr := slopeRetr / fRampTime_s;
        fPositionReference_m := ((x4 - ((x1_tmp_0 - x1_tmp) * fVelocitySetpoint_m)) - (slopeExt * fVelocitySetpoint_m)) - ((slopeRetr * (slopeExt * slopeExt)) / 2.0);
        fVelocityReference_m := ( -fVelocitySetpoint_m) - (slopeExt * slopeRetr);
    ELSE 
        fPositionReference_m := fStartPosition_m;
        fVelocityReference_m := fStartVelocity_m;
    END_IF;
END_IF;
fTotalMotionTime_s := ((((((fTimeBeforeStarting_s + fRampTime_s) + tHold) + fRampTime_s) + fHoldPositionTime_s) + fRampTime_s) + tHold) + fRampTime_s;

(* End of Outputs for SubSystem: '<Root>/FB_MotionReferenceGenerator' *)

END_FUNCTION_BLOCK

// ---- Actuators/FBs/FB_OpenLoopWinchControl.TcPOU
FUNCTION_BLOCK FB_OpenLoopWinchControl
VAR_INPUT
	bEnable		: BOOL;
	fVelocityReference_ms: LREAL;
	stOpenLoopSettings : ST_OpenLoopParams;
END_VAR
VAR_OUTPUT
	fOutput: LREAL;
END_VAR
VAR
	fFlowReference_LpM : LREAL;
	fRads : LREAL;
	stWinchParams : ST_WinchParameters; 
END_VAR

fRads := (fVelocityReference_ms/G_Parameters.stWinchParams.fWinchDrumScaling)*3.14/180; // m/s to rad/s
//fFlowReference_lmin := (fDisplacment_cc*(fRads/(2*3.14)*60))/1000;
fFlowReference_LpM := (G_Parameters.stWinchParams.fWinchMotorDisplacement*1E-5*fRads/(2*3.14))*60000; // m^3/s to l/min

IF bEnable THEN 
    fOutput := (fFlowReference_LpM) / stOpenLoopSettings.fMaxFlow;
ELSE 
    fOutput := 0.0;
END_IF;

IF fOutput > 1.0 THEN 
    fOutput := 1.0;
ELSIF fOutput < -1.0 THEN 
    fOutput := -1.0;
END_IF;

END_FUNCTION_BLOCK

// ---- Actuators/FBs/FB_ResetIntegralController.TcPOU
FUNCTION_BLOCK FB_ResetIntegralController
VAR_INPUT
	fVelocityReference_ms: LREAL;
	fMaxPositionError_m: LREAL;
	fPositionError_m: LREAL;
END_VAR
VAR_OUTPUT
	bReset: BOOL;
END_VAR
VAR
	rtb_Reset: DINT;
END_VAR


(* Outputs for Atomic SubSystem: '<Root>/FB_ResetIntegralController' *)
(* MATLAB Function: '<S1>/ResetIntegralController' *)
(* MATLAB Function 'FB_ResetIntegralController/ResetIntegralController': '<S2>:1' *)
(* '<S2>:1:3' if abs(vRef) > 0 || abs(exCyl) > exCylMax *)

IF ABS(fVelocityReference_ms) > 0.0 THEN 
    (* '<S2>:1:4' Reset = 0; *)
    rtb_Reset := 0;
ELSIF ABS(fPositionError_m) > fMaxPositionError_m THEN 
    (* '<S2>:1:4' Reset = 0; *)
    rtb_Reset := 0;
ELSE 
    (* '<S2>:1:5' else *)
    (* '<S2>:1:6' Reset = 1; *)
    rtb_Reset := 1;
END_IF;

(* End of MATLAB Function: '<S1>/ResetIntegralController' *)


(* Outport: '<Root>/bReset' incorporates:
 *  DataTypeConversion: '<S1>/Data Type Conversion' *)
bReset := rtb_Reset <> 0;
(* End of Outputs for SubSystem: '<Root>/FB_ResetIntegralController' *)

END_FUNCTION_BLOCK

// ---- Actuators/FBs/FB_ClosedLoopControl.TcPOU
FUNCTION_BLOCK FB_ClosedLoopControl
VAR_INPUT
	bEnable: BOOL;
	bActivateIntegralController: BOOL;
	fPositionReference: LREAL;
	fPositionFeedback: LREAL;
	bIntegralControllReset: BOOL;
	stClosedLoopParams : ST_ClosedLoopParams; 
	stMotionParams : ST_MotionReferenceParams; 
END_VAR
VAR_OUTPUT
	fClosedLoopPosition: LREAL;
	fPositionError: LREAL;
END_VAR
VAR
	rtb_u_FB: LREAL;
	rtb_Saturation1: LREAL;
	c_DiscreteTimeIntegrator_DS: LREAL;
END_VAR



(* SystemInitialize for Atomic SubSystem: '<Root>/FB_ClosedLoopControl' *)
(* InitializeConditions for DiscreteIntegrator: '<S1>/Discrete-Time Integrator' *)
c_DiscreteTimeIntegrator_DS := 0.0;
(* End of SystemInitialize for SubSystem: '<Root>/FB_ClosedLoopControl' *)

(* Outputs for Atomic SubSystem: '<Root>/FB_ClosedLoopControl' *)
(* Sum: '<S1>/Sum1' *)
fPositionError := fPositionReference - fPositionFeedback;
(* DiscreteIntegrator: '<S1>/Discrete-Time Integrator' *)

IF bIntegralControllReset THEN 
	c_DiscreteTimeIntegrator_DS := 0.0;
END_IF;


IF c_DiscreteTimeIntegrator_DS >= 1.0 THEN 
	c_DiscreteTimeIntegrator_DS := 1.0;
ELSIF c_DiscreteTimeIntegrator_DS <= -1.0 THEN 
	c_DiscreteTimeIntegrator_DS := -1.0;
END_IF;

(* Switch: '<S1>/Switch' incorporates:
 *  Constant: '<S1>/Constant'
 *  DiscreteIntegrator: '<S1>/Discrete-Time Integrator' *)

IF bActivateIntegralController THEN 
	rtb_u_FB := c_DiscreteTimeIntegrator_DS;
ELSE 
	rtb_u_FB := 0.0;
END_IF;

(* End of Switch: '<S1>/Switch' *)


(* Sum: '<S1>/Sum5' incorporates:
 *  Product: '<S1>/Product' *)
rtb_u_FB := (stClosedLoopParams.fProportionalGain * fPositionError) + rtb_u_FB;
(* Saturate: '<S1>/Saturation1' *)

IF rtb_u_FB > 1.0 THEN 
	rtb_Saturation1 := 1.0;
ELSIF rtb_u_FB >= -1.0 THEN 
	rtb_Saturation1 := rtb_u_FB;
ELSE 
	rtb_Saturation1 := -1.0;
END_IF;

(* End of Saturate: '<S1>/Saturation1' *)


(* Switch: '<S1>/Switch1' *)

IF bEnable THEN 
	(* Outport: '<Root>/fClosedLoopPosition' *)
	fClosedLoopPosition := rtb_Saturation1;
ELSE 
	(* Outport: '<Root>/fClosedLoopPosition' incorporates:
	 *  Constant: '<S1>/Constant1' *)
	fClosedLoopPosition := 0.0;
END_IF;

(* End of Switch: '<S1>/Switch1' *)


(* Update for DiscreteIntegrator: '<S1>/Discrete-Time Integrator' incorporates:
 *  Product: '<S1>/Divide'
 *  Product: '<S1>/Product2'
 *  Sum: '<S1>/Sum2'
 *  Sum: '<S1>/Sum3' *)
c_DiscreteTimeIntegrator_DS := (((((rtb_Saturation1 - rtb_u_FB) / stClosedLoopParams.fProportionalGain) + fPositionError) * stClosedLoopParams.fIntegralGain) * stMotionParams.fCycleTime) + c_DiscreteTimeIntegrator_DS;

IF c_DiscreteTimeIntegrator_DS >= 1.0 THEN 
	c_DiscreteTimeIntegrator_DS := 1.0;
ELSIF c_DiscreteTimeIntegrator_DS <= -1.0 THEN 
	c_DiscreteTimeIntegrator_DS := -1.0;
END_IF;

(* End of Update for DiscreteIntegrator: '<S1>/Discrete-Time Integrator' *)
(* End of Outputs for SubSystem: '<Root>/FB_ClosedLoopControl' *)

END_FUNCTION_BLOCK

// ---- Actuators/FBs/FB_AutoCyl.TcPOU
FUNCTION_BLOCK FB_AutoCyl
VAR_INPUT
	bEnable 							: BOOL;
	bStartMotion 						: BOOL;
	bStopMotion 						: BOOL;
	stMotionRefGenerator : ST_MotionReferenceParams;
	stClosedLoopControl : ST_ClosedLoopParams;
	stOpenLoopControl : ST_OpenLoopParams;
	stControlSelect			: ST_AutoControllerSelection;
	stScaledValues : ST_ScalingParameters;
	stScaledWinch : ST_WinchParameters;  
	fPositionFeedback					: LREAL;
END_VAR
VAR_OUTPUT
	fTime : LREAL;
	fVelocityReference_ms : LREAL;
	fPositionReference_m : LREAL;
	fControlOutputNormalized : LREAL;
	fPositionError_mm : LREAL;
END_VAR
VAR
	fbClock : FB_Timer;	
	fbMotionReferenceGenerator 		: FB_MotionReferenceGenerator;	
	fbFeedForwardControl 	: FB_OpenLoopControlCyl;
	fbResetIntegralController 		: FB_ResetIntegralController; 
	fbClosedLoopControl 	: FB_ClosedLoopControl;
END_VAR

fbClock(
	bEnable := bEnable,
	bStart := bStartMotion,
	bStop := bStopMotion,
	fCycleTime := stMotionRefGenerator.fCycleTime);

fbMotionReferenceGenerator(
	bEnable := bEnable,
	stMotionParameters := stMotionRefGenerator,
	fClock_s := fbClock.fTime
);

fbFeedForwardControl(
	bEnable := stControlSelect.bStartFeedForward,
	fVelocityReference_ms := fbMotionReferenceGenerator.fVelocityReference_m,
	stOpenLoopSettings := stOpenLoopControl); 
	
fbClosedLoopControl(
	bEnable := stControlSelect.bStartClosedLoop,
	bActivateIntegralController := stControlSelect.bEnableIntegral,
	fPositionReference := fbMotionReferenceGenerator.fPositionReference_m,
	fPositionFeedback := fPositionFeedback,
	bIntegralControllReset := fbResetIntegralController.bReset,
	stClosedLoopParams := stClosedLoopControl,
	stMotionParams := stMotionRefGenerator
	
); 

fbResetIntegralController(
	fMaxPositionError_m := stClosedLoopControl.fMaxAllowableError,
	fPositionError_m := fbClosedLoopControl.fPositionError,
	fVelocityReference_ms := fbMotionReferenceGenerator.fVelocityReference_m
	
); 


fVelocityReference_ms := fbMotionReferenceGenerator.fVelocityReference_m;
fPositionReference_m := fbMotionReferenceGenerator.fPositionReference_m;
fTime := fbClock.fTime;
fPositionError_mm := fbClosedLoopControl.fPositionError*1E3; 

IF bEnable THEN
	fControlOutputNormalized := LIMIT(-1.0, (fbFeedForwardControl.fVelocityFeedForward + fbClosedLoopControl.fClosedLoopPosition), 1.0); 
ELSE
	fControlOutputNormalized := 0.0; 
END_IF

END_FUNCTION_BLOCK

// ---- Actuators/FBs/FB_OpenLoopControlCyl.TcPOU
FUNCTION_BLOCK FB_OpenLoopControlCyl
VAR_INPUT
	bEnable: BOOL;
	fVelocityReference_ms: LREAL;
	stOpenLoopSettings : ST_OpenLoopParams;
END_VAR
VAR_OUTPUT
	fVelocityFeedForward: LREAL;
END_VAR
VAR
	fFlowReference : LREAL;
END_VAR


(* Outputs for Atomic SubSystem: '<Root>/FB_OpenLoopControl' *)
(* Switch: '<S1>/Switch2' incorporates:
 *  Constant: '<S1>/Annnulus_Area'
 *  Constant: '<S1>/Bore_Area'
 *  Product: '<S1>/Product1'
 *  Product: '<S1>/Product3' *)

IF fVelocityReference_ms >= 0.0 THEN 
    fFlowReference := stOpenLoopSettings.fBoresideArea * fVelocityReference_ms; // Generates flow to bore side
ELSE 
    fFlowReference := fVelocityReference_ms * stOpenLoopSettings.fAnnulusArea; // Generates flow to piston side (Q=A*v)
END_IF;

(* End of Switch: '<S1>/Switch2' *)


(* Switch: '<S1>/Switch1' incorporates:
 *  Constant: '<S1>/Constant'
 *  Gain: '<S1>/Gain1'
 *  Product: '<S1>/Divide2' *)

IF bEnable THEN 
    fVelocityFeedForward := (60000.0 * fFlowReference) / stOpenLoopSettings.fMaxFlow;
ELSE 
    fVelocityFeedForward := 0.0;
END_IF;

(* End of Switch: '<S1>/Switch1' *)


(* Saturate: '<S1>/Saturation1' *)

IF fVelocityFeedForward > 1.0 THEN 
    (* Outport: '<Root>/fVelocityFeedForward' *)
    fVelocityFeedForward := 1.0;
ELSIF fVelocityFeedForward < -1.0 THEN 
    (* Outport: '<Root>/fVelocityFeedForward' *)
    fVelocityFeedForward := -1.0;
END_IF;

(* End of Saturate: '<S1>/Saturation1' *)
(* End of Outputs for SubSystem: '<Root>/FB_OpenLoopControl' *)

END_FUNCTION_BLOCK

// ---- HMI/FBs/FB_Status.TcPOU
FUNCTION_BLOCK FB_Status
VAR_INPUT
	bFault : BOOL;
	bStart : BOOL;
	bStop : BOOL;
	bRunning : BOOL;
	bAuto : BOOL;
	bOn : BOOL;
END_VAR
VAR_OUTPUT
	eStatus : E_Status := E_Status.NotReady;
END_VAR
VAR
END_VAR


CASE eStatus OF 

	E_Status.NotReady:
		IF bOn THEN
			eStatus := E_Status.Ready;
		ELSE
			G_Modes.stVisualParams.bFault := FALSE;
			G_Modes.stVisualParams.bStop := FALSE;
			eStatus := E_Status.NotReady;
			
			
		END_IF
		
	E_Status.Ready:
		IF bOn THEN
			eStatus := E_Status.Ready;
		ELSE
			eStatus := E_Status.NotReady;
		END_IF
		
		IF bStart THEN
			eStatus := E_Status.Starting;
		END_IF
	
	E_Status.Starting:
			eStatus := E_Status.Running;
		
	E_Status.Running:
		IF bAuto AND bStart AND bOn THEN
			G_Modes.stVisualParams.bRunning := TRUE;
			eStatus := E_Status.Running;
			
		ELSIF
			bFault THEN
			eStatus := E_Status.Fault;
			
		ELSIF
			 NOT (bAuto) AND bOn THEN
			G_Modes.stVisualParams.bRunning := TRUE;
			eStatus := E_Status.Running;
				IF bStop THEN
				eStatus := E_Status.Stopping;
				END_IF
		
		
		ELSE
			G_Modes.stVisualParams.bRunning := FALSE;
			eStatus := E_Status.Ready;
		END_IF
		
		
		
		
	E_Status.Stopping:
		G_Modes.stVisualParams.bRunning := FALSE;
		bStop := TRUE;
		//Set in a delay to show the stopping longer.
		eStatus := E_Status.NotReady;
	
	E_Status.Fault:
		//Til steget der vi dektekterer fault//eStatus := E_Status.Fault;
		IF bOn THEN	
			G_Modes.stVisualParams.bStop := TRUE; // LIGHT
			G_Modes.stVisualParams.bRunning := FALSE;
			eStatus := E_Status.Fault;
		ELSE
			eStatus := E_Status.NotReady;
		END_IF
END_CASE

END_FUNCTION_BLOCK

// ---- GlobalTextList.TcGTLO
TEXTLIST GlobalTextList
  667 = 'Auto / Manual'
  369 = 'Control'
  682 = 'Current Error: %f'
  244 = 'Current Setpoint: %0.1f'
  628 = 'Cylinder Position'
  31 = 'Cylinder Position: %f'
  107 = 'CylinderPosition: %f [m]'
  78 = 'Enable Cylinder'
  609 = 'Enable WInch'
  459 = 'Engage CL'
  878 = 'Engage OL'
  106 = 'I_Gain: %0.1f'
  674 = 'I_Gain_CL: %0.1f'
  850 = 'I_Gain_OL: %0.1f'
  703 = 'Joy_X'
  91 = 'Joy_x'
  757 = 'Joy_Y'
  396 = 'MODE'
  50 = 'Mode: %s'
  270 = 'ON / OFF'
  6 = 'Piston Pressure: %f [bar]'
  891 = 'Pressure: %f [bar]'
  577 = 'P_Gain: %0.1f'
  849 = 'P_Gain_CL: %0.1f'
  155 = 'P_Gain_OL: %0.1f'
  759 = 'Return Pressure: %f [bar]'
  631 = 'Rod Pressure: %f [bar]'
  160 = 'Running'
  257 = 'Sensor Readings'
  83 = 'Start'
  655 = 'Start integrator'
  882 = 'Status : %s'
  80 = 'Stop'
  880 = 'Stopping / Fault'
  673 = 'Supply Pressure: %f [bar]'
  74 = 'VRBHMI'
  662 = 'WinchDrainPressure: %f [bar]'
  694 = 'WinchEnable'
  633 = 'WinchFlow: %f [L/Min]'
  787 = 'WinchOnly'
  786 = 'Winch_A1_Pressure: %f [bar]'
  835 = 'Winch_A_Pressure: %f [bar]'
  574 = 'Winch_B1_Pressure: %f [bar]'
  905 = 'Winch_B_Pressure: %f [bar]'
  370 = 'Wire Position'
  918 = 'Wire Position: %f'
  744 = 'Wire Position: %f [m]'
END_TEXTLIST

// ---- HMI/CtrlBox.TcVIS
VISUALIZATION CtrlBox  // 2x2
END_VISUALIZATION

// ---- HMI/VirtualBoxHMI.TcVIS
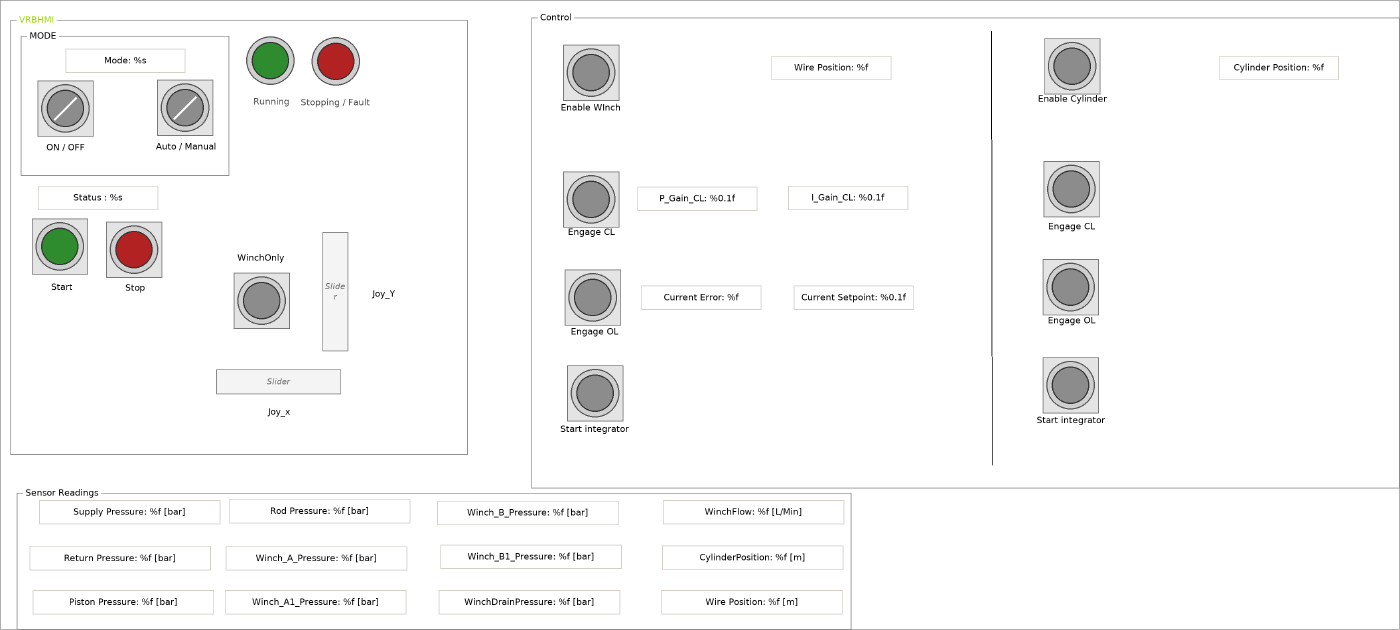
VISUALIZATION VirtualBoxHMI  // 1755x790
    GroupBox (13,17 573x553), "VRBHMI"
        PushSwitch (27,257 70x70), variable: G_Modes.bStart, behaviour: TAP, style: Switch-PushSwitch-Green
        PushSwitch (120,261 70x70), variable: G_Modes.bStop, behaviour: TAP, style: Switch-PushSwitch-Red
        Lamp1 (291,24 70x70), variable: G_Modes.stVisualParams.bRunning, style: Lamp-Lamp1-Green
        Lamp1 (373,25 70x70), variable: G_Modes.stVisualParams.bStop, style: Lamp-Lamp1-Red
        Slider (5682,5127 161x29), scale 0..100
        Slider (5815,4955 30x143), scale 0..100
        Label (5690,5182 150x30), "Joy_X"
        Label (5852,4969 65x118), "Joy_Y"
        Label (360,97 95x29), "Stopping / Fault"
        Label (105,330 103x28), "Stop"
        Label (19,328 91x30), "Start"
        GroupBox (13,20 261x183), "MODE"
            Label (11,133 91x30), "ON / OFF"
            RotarySwitch (171,63 70x70), variable: G_Modes.bAutoMode, behaviour: TOGGLE, style: Switch-RotarySwitch-Gray
            Label (162,132 91x30), "Auto / Manual"
            Textfield (56,24 150x30), "Mode: %s", text variable: G_Modes.eMode
            RotarySwitch (21,64 70x70), variable: G_Modes.bOn, behaviour: TOGGLE, style: Switch-RotarySwitch-Gray
        Textfield (35,216 150x30), "Status : %s", text variable: G_Modes.eStatus
        Label (193,329 103x28)
        Label (280,96 95x29), "Running"
        Slider (258,446 156x31), variable: G_InputsScaled.fJoystickScaledX, scale -1..1
        Slider (391,274 32x149), variable: G_InputsScaled.fJoystickScaledY, scale -1..1
        Label (298,484 78x31), "Joy_x"
        Label (433,338 70x27), "Joy_Y"
        PushSwitch (280,325 70x70), variable: G_Modes.bSwitch, behaviour: TOGGLE, style: Switch-PushSwitch-Gray
        Label (279,293 70x27), "WinchOnly"
    GroupBox (666,14 1089x598), "Control"
        PushSwitch (40,42 70x70), variable: G_Modes.bWinchEnable, behaviour: TOGGLE, style: Switch-PushSwitch-Gray
        Label (29,106 91x30), "Enable WInch"
        PushSwitch (643,34 70x70), variable: G_Modes.bCylEnable, behaviour: TOGGLE, style: Switch-PushSwitch-Gray
        Label (633,95 91x30), "Enable Cylinder"
        PushSwitch (40,201 70x70), variable: G_Modes.stWinchControl.bStartClosedLoop, behaviour: TOGGLE, style: Switch-PushSwitch-Gray
        PushSwitch (42,324 70x70), variable: G_Modes.stWinchControl.bStartFeedForward, behaviour: TOGGLE, style: Switch-PushSwitch-Gray
        PushSwitch (45,444 70x70), variable: G_Modes.stWinchControl.bEnableIntegral, behaviour: TOGGLE, style: Switch-PushSwitch-Gray
        PushSwitch (642,188 70x70), variable: G_Modes.stCylinderControl.bStartClosedLoop, behaviour: TOGGLE, style: Switch-PushSwitch-Gray
        PushSwitch (641,311 70x70), variable: G_Modes.stCylinderControl.bStartFeedForward, behaviour: TOGGLE, style: Switch-PushSwitch-Gray
        PushSwitch (641,434 70x70), variable: G_Modes.stCylinderControl.bEnableIntegral, behaviour: TOGGLE, style: Switch-PushSwitch-Gray
        Label (30,262 91x30), "Engage CL"
        Label (632,255 91x30), "Engage CL"
        Label (34,387 91x30), "Engage OL"
        Label (632,373 91x30), "Engage OL"
        Label (34,509 91x30), "Start integrator"
        Label (631,498 91x30), "Start integrator"
        Line (578,569) (577,25)
        Textfield (301,56 150x30), "Wire Position: %f", text variable: G_InputsScaled.fWirePosition
        Textfield (862,56 150x30), "Cylinder Position: %f", text variable: G_InputsScaled.fCylPosition
        Textfield (133,220 150x30), "P_Gain_CL: %0.1f", text variable: G_Parameters.stControl.stCylControlCloesSettings.fProportionalGain
        Textfield (322,219 150x30), "I_Gain_CL: %0.1f", text variable: G_Parameters.stControl.stCylControlCloesSettings.fIntegralGain
        Textfield (138,344 150x30), "Current Error: %f", text variable: G_ControlParameters.fPosErrorWinch
        Textfield (329,344 150x30), "Current Setpoint: %0.1f", text variable: G_ControlParameters.fVelRefWinch
    GroupBox (21,610 1046x180), "Sensor Readings"
        Textfield (28,17 227x30), "Supply Pressure: %f [bar]", text variable: G_InputsScaled.fSupplyPressure
        Textfield (266,16 227x30), "Rod Pressure: %f [bar]", text variable: G_InputsScaled.fRodPressure
        Textfield (262,75 227x30), "Winch_A_Pressure: %f [bar]", text variable: G_InputsScaled.fWinch_A_Pressure
        Textfield (261,130 227x30), "Winch_A1_Pressure: %f [bar]", text variable: G_InputsScaled.fWinch_A1_Pressure
        Textfield (527,18 227x30), "Winch_B_Pressure: %f [bar]", text variable: G_InputsScaled.fWinch_B_Pressure
        Textfield (531,73 227x30), "Winch_B1_Pressure: %f [bar]", text variable: G_InputsScaled.fWinch_B1_Pressure
        Textfield (529,130 227x30), "WinchDrainPressure: %f [bar]", text variable: G_InputsScaled.fWinchDrainPressure
        Textfield (808,130 227x30), "Wire Position: %f [m]", text variable: G_InputsScaled.fWirePosition
        Textfield (809,74 227x30), "CylinderPosition: %f [m]", text variable: G_InputsScaled.fCylPosition
        Textfield (810,17 227x30), "WinchFlow: %f [L/Min]", text variable: G_InputsScaled.fWinchFlow
        Textfield (16,75 227x30), "Return Pressure: %f [bar]", text variable: G_InputsScaled.fReturnPressure
        Textfield (20,130 227x30), "Piston Pressure: %f [bar]", text variable: G_InputsScaled.fPistonPressure
END_VISUALIZATION
